FUNCTION F_InitializeAllGroups :BOOL
(**************************************************************************************
 * 	Application		:	BoxControl Framework
 *	Revision		:	$Revision: 404529 $
 *	Revision date	:	$Date: 2018-04-23 08:21:38 +0200 (Mo., 23 Apr 2018) $
 *	Last changed by	:	$Author: b7bolm $
 *	URL				:	$URL: http://almscdc.swisslog.com/repo/SWPD/Development/BoxControlFramework/20_Release/trunk/01_Software/BCF/BCF/JumpStart/20_Product/10_App/14_Groups/10_Lib/10_Conv/10_Functions/F_InitializeAllGroups.TcPOU $
 *
 *	Purpose			:	Initialize all groups
 *
 * ------------------------------------------------------------------------------------
 *	Copyright Swisslog [IP AG], Switzerland. All rights reserved.
 * 
 * ------------------------------------------------------------------------------------
 *	
 * 	Revision History: 
 *
 * 	VERSION			DATE			INITIALS			DESCRIPTION
 *	0.1				01.01.2001		swl					Example
 *
 **************************************************************************************)
VAR
	eGroupNumber		: E_GroupNumber; // Group number
END_VAR


// Loop over all elements and initialize each group 
FOR eGroupNumber := E_GroupNumber.G_BEGIN_GROUP + 1 TO E_GroupNumber.G_END_GROUP - 1 DO
	// If reference is valid
	IF __ISVALIDREF(GroupRegistry[eGroupNumber].rGroup) THEN
		// Initialize group
		GroupRegistry[eGroupNumber].rGroup.M_InitGroup(TRUE);
	END_IF
END_FOR

END_FUNCTION

(* stored: Version 1.1.0.1, ProductVersion 3.1.4022.12
   POU F_InitializeAllGroups: Id {caeab955-f22e-4e11-9fe3-7a4fa761f02e}, SpecialFunc None *)
